(* IEC 61131-3 sources: Word/plc-course/14-analog-and-process-io/labs/solutions, 3 files *)

(* ---- 14-1-analog-input.st ---- *)
(* Lab 14-1: FB_AnalogInput - raw counts to engineering units, with
   NAMUR NE43 fault detection, clamping, a first-order filter, a quality
   flag and substitute-value behaviour.
   Module 14 (Analog signals and process I/O). REFERENCE SOLUTION - try the lab yourself first.

   Raw-count convention used by every lab in this module (Siemens style):
     Raw = 0     ->  4 mA   (bottom of the rated range)
     Raw = 27648 -> 20 mA   (top of the rated range)
     1 mA = 27648 / 16 = 1728 counts.
   Values outside 0..27648 are under- and over-range. The simulated card
   in this lab is linear over the whole INT range, so 0 mA reads -6912 and
   21 mA reads 29376. The Siemens underflow/overflow codes (-32768, 32767)
   also land in the failure bands, so this block copes with them too. *)

FUNCTION_BLOCK FB_AnalogInput
  VAR_INPUT
    Raw        : INT;    (* raw count from the input card *)
    EuMin      : REAL;   (* engineering value at 4 mA (must be below EuMax) *)
    EuMax      : REAL;   (* engineering value at 20 mA *)
    FilterTime : TIME;   (* first-order filter time constant; T#0s = no filter *)
    FaultDelay : TIME;   (* signal must stay in a failure band this long before Fault *)
    UseSubst   : BOOL;   (* on Fault: TRUE = output SubstValue, FALSE = hold last good value *)
    SubstValue : REAL;   (* substitute value, engineering units *)
    CycleTime  : TIME;   (* interval of the task that calls this block *)
  END_VAR
  VAR_OUTPUT
    Current_mA : REAL;   (* loop current worked out from Raw: not filtered, not clamped *)
    Value      : REAL;   (* engineering value for the rest of the program *)
    Good       : BOOL;   (* TRUE while the loop current is inside the NE43 limits *)
    UnderRange : BOOL;   (* current <= 3.6 mA for FaultDelay: wire break, failure low *)
    OverRange  : BOOL;   (* current >= 21.0 mA for FaultDelay: short circuit, failure high *)
    Fault      : BOOL;   (* UnderRange OR OverRange *)
  END_VAR
  VAR CONSTANT
    COUNTS_PER_MA : REAL := 1728.0;   (* 27648 counts / 16 mA *)
    FAIL_LOW_MA   : REAL := 3.6;      (* NE43: at or below = failure signal *)
    FAIL_HIGH_MA  : REAL := 21.0;     (* NE43: at or above = failure signal *)
  END_VAR
  VAR
    LowTimer    : TON;    (* confirmation delay for the low failure band *)
    HighTimer   : TON;    (* confirmation delay for the high failure band *)
    Scaled      : REAL;   (* engineering value, clamped, before the filter *)
    Filtered    : REAL;   (* filter state; also the last good value *)
    FilterReady : BOOL;   (* FALSE until Filtered holds a real measurement *)
    Alpha       : REAL;   (* filter weight for this scan, 0..1 *)
  END_VAR

  (* 1. Raw count -> loop current. Convert to REAL before doing any
        arithmetic: Raw * 16 in INT would overflow above 2047 counts. *)
  Current_mA := 4.0 + INT_TO_REAL(Raw) / COUNTS_PER_MA;

  (* 2. NAMUR NE43 check. Each failure band has its own timer, so the
        signal must stay in the band for the whole FaultDelay. The flags
        clear on the first scan the current is back inside the limits. *)
  LowTimer(IN := Current_mA <= FAIL_LOW_MA, PT := FaultDelay);
  HighTimer(IN := Current_mA >= FAIL_HIGH_MA, PT := FaultDelay);
  UnderRange := LowTimer.Q;
  OverRange := HighTimer.Q;
  Fault := UnderRange OR OverRange;

  (* Good = the reading is a live measurement right now. It drops at once,
     without waiting for the delay; Fault is the confirmed version. *)
  Good := (Current_mA > FAIL_LOW_MA) AND (Current_mA < FAIL_HIGH_MA);

  (* 3. Linear scaling 4..20 mA -> EuMin..EuMax, then clamp. Between
        3.6 and 4 mA (and 20 and 21 mA) the reading is still trusted
        but is shown as the end of the range. *)
  Scaled := EuMin + (Current_mA - 4.0) * (EuMax - EuMin) / 16.0;
  Scaled := LIMIT(EuMin, Scaled, EuMax);

  (* 4. First-order lag filter, only fed with good readings. While the
        signal is suspect or faulted, Filtered is left alone, so it holds
        the last good value. *)
  IF Good THEN
    IF NOT FilterReady THEN
      (* First good reading after power-up or after a fault: start the
         filter here instead of ramping up from 0 or from a held value. *)
      Filtered := Scaled;
      FilterReady := TRUE;
    ELSE
      (* Alpha = Ts / (Tf + Ts). A ratio of two times has no unit, so it
         works whatever unit TIME_TO_REAL uses on your platform.
         FilterTime = T#0s gives Alpha = 1: no filtering, no division by 0. *)
      IF FilterTime > T#0s THEN
        Alpha := TIME_TO_REAL(CycleTime) / (TIME_TO_REAL(CycleTime) + TIME_TO_REAL(FilterTime));
      ELSE
        Alpha := 1.0;
      END_IF;
      Filtered := Filtered + Alpha * (Scaled - Filtered);
    END_IF;
  END_IF;

  IF Fault THEN
    FilterReady := FALSE;   (* restart the filter from the live value on recovery *)
  END_IF;

  (* 5. Output: substitute on a confirmed fault if configured, otherwise
        the filter state (live value, or the held last good value). *)
  IF Fault AND UseSubst THEN
    Value := SubstValue;
  ELSE
    Value := Filtered;
  END_IF;
END_FUNCTION_BLOCK

PROGRAM AnalogInputs
  VAR (* I/O - analog inputs, 0..27648 = 4..20 mA *)
    LT101_Raw AT %IW0 : INT;  (* LT-101 tank level transmitter: 0.0..4.0 m *)
    TT102_Raw AT %IW1 : INT;  (* TT-102 reactor temperature transmitter: -50..150 degC *)
  END_VAR
  VAR
    LT101 : FB_AnalogInput;   (* level: filtered, holds the last good value on a fault *)
    TT102 : FB_AnalogInput;   (* temperature: unfiltered, substitutes 150 degC on a fault *)
  END_VAR

  (* Level: 2 s filter to calm a surface that ripples, hold last value on a
     fault (the level alarms in Lab 14-2 then freeze rather than jump). *)
  LT101(Raw := LT101_Raw, EuMin := 0.0, EuMax := 4.0,
        FilterTime := T#2s, FaultDelay := T#1s,
        UseSubst := FALSE, SubstValue := 0.0, CycleTime := T#10ms);

  (* Temperature: no filter (a trip needs the fastest response), and a
     substitute value at the TOP of the range, so a failed transmitter
     drives a high-temperature trip rather than hiding a real overheat. *)
  TT102(Raw := TT102_Raw, EuMin := -50.0, EuMax := 150.0,
        FilterTime := T#0s, FaultDelay := T#2s,
        UseSubst := TRUE, SubstValue := 150.0, CycleTime := T#10ms);
END_PROGRAM

CONFIGURATION Config0
  RESOURCE Res0 ON PLC
    TASK MainTask(INTERVAL := T#10ms, PRIORITY := 0);
    PROGRAM Inst0 WITH MainTask : AnalogInputs;
  END_RESOURCE
END_CONFIGURATION

(* ---- 14-2-analog-alarm.st ---- *)
(* Lab 14-2: FB_AnalogAlarm - HH/H/L/LL process alarms with a deadband
   (hysteresis) and an on-delay, so a noisy signal cannot make them chatter.
   Module 14 (Analog signals and process I/O). REFERENCE SOLUTION - try the lab yourself first.

   Design: one small block, FB_LimitAlarm, handles a single limit. The
   analog alarm block uses four instances of it. MATIEC cannot make an
   array of FB instances, so they are four separate variables. *)

FUNCTION_BLOCK FB_LimitAlarm
  VAR_INPUT
    PV         : REAL;  (* process value, engineering units *)
    LimitValue : REAL;  (* alarm limit ("Limit" would clash with the LIMIT function) *)
    Deadband   : REAL;  (* how far back inside the limit the PV must go to clear *)
    OnDelay    : TIME;  (* how long the PV must stay beyond the limit to raise *)
    HighAlarm  : BOOL;  (* TRUE: alarm above the limit; FALSE: alarm below it *)
  END_VAR
  VAR_OUTPUT
    Active     : BOOL;  (* alarm condition is active *)
  END_VAR
  VAR
    DelayTimer : TON;
    Beyond     : BOOL;  (* PV is at or beyond the limit right now *)
    Returned   : BOOL;  (* PV is back inside the limit by more than the deadband *)
  END_VAR

  IF HighAlarm THEN
    Beyond := PV >= LimitValue;
    Returned := PV < LimitValue - Deadband;
  ELSE
    Beyond := PV <= LimitValue;
    Returned := PV > LimitValue + Deadband;
  END_IF;

  (* The timer runs only while the PV is beyond the limit. Any return
     inside the limit resets it, so the delay always means "continuously
     beyond the limit for OnDelay". *)
  DelayTimer(IN := Beyond, PT := OnDelay);

  (* Raise after the delay; clear at once, but only when the PV has come
     back through the deadband. In between, keep the previous state: that
     is the hysteresis. *)
  IF DelayTimer.Q THEN
    Active := TRUE;
  ELSIF Returned THEN
    Active := FALSE;
  END_IF;
END_FUNCTION_BLOCK

FUNCTION_BLOCK FB_AnalogAlarm
  VAR_INPUT
    PV       : REAL;   (* process value, engineering units *)
    HH_Limit : REAL;   (* high-high limit *)
    H_Limit  : REAL;   (* high limit *)
    L_Limit  : REAL;   (* low limit *)
    LL_Limit : REAL;   (* low-low limit *)
    Deadband : REAL;   (* engineering units, the same for all four limits *)
    OnDelay  : TIME;   (* the same for all four limits; each has its own timer *)
  END_VAR
  VAR_OUTPUT
    HH : BOOL;         (* PV >= HH_Limit for OnDelay; clears below HH_Limit - Deadband *)
    H  : BOOL;         (* PV >= H_Limit  for OnDelay; clears below H_Limit  - Deadband *)
    L  : BOOL;         (* PV <= L_Limit  for OnDelay; clears above L_Limit  + Deadband *)
    LL : BOOL;         (* PV <= LL_Limit for OnDelay; clears above LL_Limit + Deadband *)
  END_VAR
  VAR
    HH_Check : FB_LimitAlarm;
    H_Check  : FB_LimitAlarm;
    L_Check  : FB_LimitAlarm;
    LL_Check : FB_LimitAlarm;
  END_VAR

  HH_Check(PV := PV, LimitValue := HH_Limit, Deadband := Deadband, OnDelay := OnDelay, HighAlarm := TRUE);
  H_Check(PV := PV, LimitValue := H_Limit, Deadband := Deadband, OnDelay := OnDelay, HighAlarm := TRUE);
  L_Check(PV := PV, LimitValue := L_Limit, Deadband := Deadband, OnDelay := OnDelay, HighAlarm := FALSE);
  LL_Check(PV := PV, LimitValue := LL_Limit, Deadband := Deadband, OnDelay := OnDelay, HighAlarm := FALSE);

  (* The alarms are independent: at a very high PV both H and HH are
     active. Suppressing H while HH is on is an HMI or alarm-system
     decision (Module 16), not something to bury in the logic. *)
  HH := HH_Check.Active;
  H := H_Check.Active;
  L := L_Check.Active;
  LL := LL_Check.Active;
END_FUNCTION_BLOCK

PROGRAM AlarmDemo
  VAR (* process values: in a real program these come from FB_AnalogInput
         (Lab 14-1). Here the test writes them directly. *)
    Level    : REAL;   (* LT-201 tank level, % *)
    Pressure : REAL;   (* PT-202 header pressure, bar *)
  END_VAR
  VAR
    LevelAlm : FB_AnalogAlarm;
    PressAlm : FB_AnalogAlarm;
  END_VAR

  (* Level: 2 % deadband, 3 s delay - a sloshing surface must not chatter. *)
  LevelAlm(PV := Level, HH_Limit := 90.0, H_Limit := 80.0, L_Limit := 20.0, LL_Limit := 10.0,
           Deadband := 2.0, OnDelay := T#3s);

  (* Pressure: 0.2 bar deadband, no delay. *)
  PressAlm(PV := Pressure, HH_Limit := 8.0, H_Limit := 7.0, L_Limit := 2.0, LL_Limit := 1.0,
           Deadband := 0.2, OnDelay := T#0s);
END_PROGRAM

CONFIGURATION Config0
  RESOURCE Res0 ON PLC
    TASK MainTask(INTERVAL := T#10ms, PRIORITY := 0);
    PROGRAM Inst0 WITH MainTask : AlarmDemo;
  END_RESOURCE
END_CONFIGURATION

(* ---- 14-3-sump-pump.st ---- *)
(* Lab 14-3: Sump pump level control - a pump-down on/off controller with
   hysteresis, a high-level alarm, an independent low-low float for dry-run
   protection, pump fault handling, and a level-transmitter fault.
   Module 14 (Analog signals and process I/O). REFERENCE SOLUTION - try the lab yourself first.

   TRAINING EXERCISE ONLY. The low-low float trip here is ordinary control
   logic in a standard PLC, not a designed safety function (Module 20).

   Raw-count convention: 0..27648 = 4..20 mA, 1728 counts per mA.
   LT-301 range 0.0..4.0 m, so 1 m = 6912 counts.

   FB_AnalogInput below is copied unchanged from the Lab 14-1 solution. In a
   real project it would live in a library; MATIEC compiles one file, so
   the lab keeps a copy here. *)

FUNCTION_BLOCK FB_AnalogInput
  VAR_INPUT
    Raw        : INT;    (* raw count from the input card *)
    EuMin      : REAL;   (* engineering value at 4 mA (must be below EuMax) *)
    EuMax      : REAL;   (* engineering value at 20 mA *)
    FilterTime : TIME;   (* first-order filter time constant; T#0s = no filter *)
    FaultDelay : TIME;   (* signal must stay in a failure band this long before Fault *)
    UseSubst   : BOOL;   (* on Fault: TRUE = output SubstValue, FALSE = hold last good value *)
    SubstValue : REAL;   (* substitute value, engineering units *)
    CycleTime  : TIME;   (* interval of the task that calls this block *)
  END_VAR
  VAR_OUTPUT
    Current_mA : REAL;   (* loop current worked out from Raw: not filtered, not clamped *)
    Value      : REAL;   (* engineering value for the rest of the program *)
    Good       : BOOL;   (* TRUE while the loop current is inside the NE43 limits *)
    UnderRange : BOOL;   (* current <= 3.6 mA for FaultDelay: wire break, failure low *)
    OverRange  : BOOL;   (* current >= 21.0 mA for FaultDelay: short circuit, failure high *)
    Fault      : BOOL;   (* UnderRange OR OverRange *)
  END_VAR
  VAR CONSTANT
    COUNTS_PER_MA : REAL := 1728.0;   (* 27648 counts / 16 mA *)
    FAIL_LOW_MA   : REAL := 3.6;      (* NE43: at or below = failure signal *)
    FAIL_HIGH_MA  : REAL := 21.0;     (* NE43: at or above = failure signal *)
  END_VAR
  VAR
    LowTimer    : TON;    (* confirmation delay for the low failure band *)
    HighTimer   : TON;    (* confirmation delay for the high failure band *)
    Scaled      : REAL;   (* engineering value, clamped, before the filter *)
    Filtered    : REAL;   (* filter state; also the last good value *)
    FilterReady : BOOL;   (* FALSE until Filtered holds a real measurement *)
    Alpha       : REAL;   (* filter weight for this scan, 0..1 *)
  END_VAR

  (* 1. Raw count -> loop current. Convert to REAL before doing any
        arithmetic: Raw * 16 in INT would overflow above 2047 counts. *)
  Current_mA := 4.0 + INT_TO_REAL(Raw) / COUNTS_PER_MA;

  (* 2. NAMUR NE43 check. Each failure band has its own timer, so the
        signal must stay in the band for the whole FaultDelay. The flags
        clear on the first scan the current is back inside the limits. *)
  LowTimer(IN := Current_mA <= FAIL_LOW_MA, PT := FaultDelay);
  HighTimer(IN := Current_mA >= FAIL_HIGH_MA, PT := FaultDelay);
  UnderRange := LowTimer.Q;
  OverRange := HighTimer.Q;
  Fault := UnderRange OR OverRange;

  (* Good = the reading is a live measurement right now. It drops at once,
     without waiting for the delay; Fault is the confirmed version. *)
  Good := (Current_mA > FAIL_LOW_MA) AND (Current_mA < FAIL_HIGH_MA);

  (* 3. Linear scaling 4..20 mA -> EuMin..EuMax, then clamp. Between
        3.6 and 4 mA (and 20 and 21 mA) the reading is still trusted
        but is shown as the end of the range. *)
  Scaled := EuMin + (Current_mA - 4.0) * (EuMax - EuMin) / 16.0;
  Scaled := LIMIT(EuMin, Scaled, EuMax);

  (* 4. First-order lag filter, only fed with good readings. While the
        signal is suspect or faulted, Filtered is left alone, so it holds
        the last good value. *)
  IF Good THEN
    IF NOT FilterReady THEN
      (* First good reading after power-up or after a fault: start the
         filter here instead of ramping up from 0 or from a held value. *)
      Filtered := Scaled;
      FilterReady := TRUE;
    ELSE
      (* Alpha = Ts / (Tf + Ts). A ratio of two times has no unit, so it
         works whatever unit TIME_TO_REAL uses on your platform.
         FilterTime = T#0s gives Alpha = 1: no filtering, no division by 0. *)
      IF FilterTime > T#0s THEN
        Alpha := TIME_TO_REAL(CycleTime) / (TIME_TO_REAL(CycleTime) + TIME_TO_REAL(FilterTime));
      ELSE
        Alpha := 1.0;
      END_IF;
      Filtered := Filtered + Alpha * (Scaled - Filtered);
    END_IF;
  END_IF;

  IF Fault THEN
    FilterReady := FALSE;   (* restart the filter from the live value on recovery *)
  END_IF;

  (* 5. Output: substitute on a confirmed fault if configured, otherwise
        the filter state (live value, or the held last good value). *)
  IF Fault AND UseSubst THEN
    Value := SubstValue;
  ELSE
    Value := Filtered;
  END_IF;
END_FUNCTION_BLOCK

PROGRAM SumpPump
  VAR (* I/O *)
    LT301_Raw     AT %IW0   : INT;   (* LT-301 sump level: 0..27648 = 4..20 mA = 0.0..4.0 m *)
    LSLL302_NC    AT %IX0.0 : BOOL;  (* low-low float, NC: TRUE while water is above it *)
    PumpRunFb     AT %IX0.1 : BOOL;  (* pump contactor auxiliary contact: TRUE = pulled in *)
    PumpOL_NC     AT %IX0.2 : BOOL;  (* motor overload relay, NC: TRUE = healthy *)
    ResetPB       AT %IX0.3 : BOOL;  (* fault reset push-button, NO *)
    PumpRun       AT %QX0.0 : BOOL;  (* pump contactor coil *)
    HighLevelAlm  AT %QX0.1 : BOOL;  (* high sump level alarm *)
    LowLowAlm     AT %QX0.2 : BOOL;  (* low-low float operated (latched) *)
    PumpFaultAlm  AT %QX0.3 : BOOL;  (* pump fault: overload or no run feedback (latched) *)
    LevelFaultAlm AT %QX0.4 : BOOL;  (* LT-301 signal outside the NE43 limits *)
  END_VAR
  VAR
    Level : REAL;                    (* sump level in m, for the HMI *)
  END_VAR
  VAR CONSTANT
    START_LEVEL    : REAL := 2.0;    (* pump starts at or above this level, m *)
    STOP_LEVEL     : REAL := 1.0;    (* pump stops at or below this level, m *)
    HIGH_ALM_LEVEL : REAL := 3.0;    (* high level alarm limit, m *)
    HIGH_ALM_DB    : REAL := 0.1;    (* high level alarm deadband, m *)
  END_VAR
  VAR
    LT301        : FB_AnalogInput;
    HighAlmTimer : TON;              (* 5 s on-delay for the high level alarm *)
    FbTimer      : TON;              (* 2 s run-feedback supervision *)
    ResetEdge    : R_TRIG;           (* reset acts on the press, not the level *)
    Demand       : BOOL;             (* the level controller wants the pump on *)
    Trip         : BOOL;             (* something stops the pump *)
  END_VAR

  (* 1. Level measurement: scaling, clamping and NE43 checking by the
        Lab 14-1 block. No filter, so the controller sees the real level.
        During the 1 s confirmation delay the block holds the last good
        level, so a broken wire does not look like an empty sump. *)
  LT301(Raw := LT301_Raw, EuMin := 0.0, EuMax := 4.0,
        FilterTime := T#0s, FaultDelay := T#1s,
        UseSubst := FALSE, SubstValue := 0.0, CycleTime := T#10ms);
  Level := LT301.Value;
  LevelFaultAlm := LT301.Fault;      (* clears by itself when the signal is healthy again *)

  (* 2. High level alarm: 5 s on-delay, 0.1 m deadband. *)
  HighAlmTimer(IN := Level >= HIGH_ALM_LEVEL, PT := T#5s);
  IF HighAlmTimer.Q THEN
    HighLevelAlm := TRUE;
  ELSIF Level < HIGH_ALM_LEVEL - HIGH_ALM_DB THEN
    HighLevelAlm := FALSE;
  END_IF;

  (* 3. Reset: one press, one reset. A jammed button cannot keep clearing
        faults and restarting a pump that keeps failing. *)
  ResetEdge(CLK := ResetPB);

  (* 4. Low-low float: independent of the transmitter, so it still protects
        the pump when LT-301 reads wrong (stuck, drifted, wrong range).
        Latched: the float should never operate in normal service, so a
        person must look before the pump runs again. The reset only works
        once the float is healthy (the IF sets it again every scan while
        the float is open). *)
  IF NOT LSLL302_NC THEN
    LowLowAlm := TRUE;
  ELSIF ResetEdge.Q THEN
    LowLowAlm := FALSE;
  END_IF;

  (* 5. Pump faults, latched until a reset:
        - overload relay tripped (reset only works once it is healthy)
        - pump commanded but no run feedback for 2 s (contactor failed to
          pull in, or dropped out while running). *)
  FbTimer(IN := PumpRun AND NOT PumpRunFb, PT := T#2s);
  IF (NOT PumpOL_NC) OR FbTimer.Q THEN
    PumpFaultAlm := TRUE;
  ELSIF ResetEdge.Q THEN
    PumpFaultAlm := FALSE;
  END_IF;

  (* 6. Pump-down level control with hysteresis. Any trip stops the pump
        at once and cancels the demand, so after a reset or recovery the
        pump starts again only when the level reaches START_LEVEL. *)
  Trip := LowLowAlm OR PumpFaultAlm OR LevelFaultAlm;

  IF Trip THEN
    Demand := FALSE;
  ELSIF Level >= START_LEVEL THEN
    Demand := TRUE;
  ELSIF Level <= STOP_LEVEL THEN
    Demand := FALSE;
  END_IF;                            (* between the two levels: keep the state *)

  PumpRun := Demand AND NOT Trip;
END_PROGRAM

CONFIGURATION Config0
  RESOURCE Res0 ON PLC
    TASK MainTask(INTERVAL := T#10ms, PRIORITY := 0);
    PROGRAM Inst0 WITH MainTask : SumpPump;
  END_RESOURCE
END_CONFIGURATION
